// TIA Portal V17 export
// export: Created 2024-08-09T12:53:05.5966737Z, ExportSetting WithDefaults, DisplayName Totally Integrated Automation Portal, DisplayVersion V17 Update 7, DisplayName TIA Portal Openness, DisplayVersion V17 Update 7, DisplayName TIA Portal Version Control Interface, DisplayVersion V17, DisplayName STEP 7 Professional, DisplayVersion V17 Update 7, DisplayName STEP 7 Safety, DisplayVersion V17 Update 6, DisplayName WinCC Professional, DisplayVersion V17 Update 7
VAR_GLOBAL   // PLC tag table "TypeCel"
END_VAR
VAR_GLOBAL CONSTANT   // user constants
   RECF1 : USInt := 16#1;
   RECF2 : USInt := 16#2;
   RECF3 : USInt := 16#4;
   RECF4 : USInt := 16#8;
   TRANSF1 : USInt := 16#10;
   VRAC : USInt := 16#20;
   ORIG_ENS1 : USInt := 16#40;
   ORIG_ENS2 : USInt := 16#80;
END_VAR
